TYPE ST_Inverter_LineState :
STRUCT
	b_LineVoltTripLimHigh		: BOOL;
	b_LineVoltTripLimlow		: BOOL;
	b_LineFreqTripLimHigh		: BOOL;
	b_LineFreqTripLimLow		: BOOL;
	b_LineFreqOK				: BOOL;
	b_LineVoltOK				: BOOL;
	b_FRTActive					: BOOL;
	b_GridCodeTripActive		: BOOL;
END_STRUCT
END_TYPE

(* stored: Version 1.1.0.1, ProductVersion 3.1.4026.18
   DUT ST_Inverter_LineState: Id {852ba63b-4727-44c5-8054-96b62b211dbe} *)
